(* IEC 61131-3 sources: inproshop/TEAM_V2.0-demo_exported/OP30/2.PRG, 7 files *)

(* ---- OP30_Communication.st ---- *)
PROGRAM OP30_Communication
VAR
	HeartdelayON:TON;
	HeartdelayOFF:TON;
	MasterHeartdelayON:TON;
	MasterHeartdelayOFF:TON;
END_VAR

//心跳输出
IF CPU_Clock.Clock_1s THEN
	DB3005_Communication.TO_OPXX.Heart:=1;
ELSE
	DB3005_Communication.TO_OPXX.Heart:=0;
END_IF
//给前站安全信号
IF TRUE THEN
	DB3005_Communication.TO_OPXX.Safe:=1;
ELSE
	DB3005_Communication.TO_OPXX.Safe:=0;
END_IF;

HeartdelayON(IN:= DB3005_Communication.From_OPXX.Heart=1, PT:= T#2S, Q=> , ET=> );
HeartdelayOFF(IN:= DB3005_Communication.From_OPXX.Heart=0, PT:= T#2S, Q=> , ET=> );
//前站掉线报警
IF (HeartdelayON.Q OR HeartdelayOFF.Q) AND NOT DB3000_Control.Mode.Status.OfflineMode  THEN
	DB3070_Fault.Stop.BeforStation_Communication_Rrror:=TRUE;
END_IF

//主站心跳通讯检测
MasterHeartdelayON(IN:= DB3005_Communication.FromMaster.Heart=1, PT:= T#2S, Q=> , ET=> );
MasterHeartdelayOFF(IN:= DB3005_Communication.FromMaster.Heart=0, PT:= T#2S, Q=> , ET=> );
//主站掉线报警
IF (MasterHeartdelayON.Q OR MasterHeartdelayOFF.Q) AND NOT DB3000_Control.Mode.Status.OfflineMode  THEN
	DB3070_Fault.Stop.MasterTimeOut:=TRUE;
END_IF

//与主站配方不一致报警
IF DB3005_Communication.FromMaster.MasterRecipeID<>DB3002_Recipe.RecipeNum AND NOT DB3000_Control.Mode.Status.OfflineMode THEN
	DB3070_Fault.Stop.MaterReipeDiscrepancy:=TRUE;
END_IF

(* ---- OP30_Control.st ---- *)
PROGRAM OP30_Control
VAR
	FB_ModeControl_instance:FB_ModeControl_V1;
	FB_Count_instance:ARRAY[0..2] OF FB_Count;
END_VAR

(**********模式切换功能***********)
FB_ModeControl_instance(
	iClock:= CPU_Clock,
	iStartDelay:= T#100MS,
	iEstop:=DB3070_Fault.EstopTotal,
	iAlam:=DB3070_Fault.StopTotal,
	iWarn:=DB3070_Fault.RunTotal,
	ioMachine:= DB3000_Control.Machine,
	ioMode:=DB3000_Control.Mode);

(********************计数****************************)
//总计数
FB_Count_instance[0](
	ioCount:= DB3003_Count.Total,
	iClock:= CPU_Clock,
	iDayStartTime:= CPU_Clock.DayStartTime,
	iNightStartTime:=CPU_Clock.NightStartTime);

//OK计数
FB_Count_instance[1](
	ioCount:= DB3003_Count.OK,
	iClock:= CPU_Clock,
	iDayStartTime:= CPU_Clock.DayStartTime,
	iNightStartTime:=CPU_Clock.NightStartTime);

//NG计数
FB_Count_instance[2](
	ioCount:= DB3003_Count.NG,
	iClock:= CPU_Clock,
	iDayStartTime:= CPU_Clock.DayStartTime,
	iNightStartTime:=CPU_Clock.NightStartTime);

(***********良率计算***********)
//良率统计
IF DB3003_Count.Total.Today.Total<>0 THEN
	DB3003_Count.Yield:=DB3003_Count.OK.Today.Total/DB3003_Count.Total.Today.Total;
ELSE
	DB3003_Count.Yield:=0;
END_IF
//良率清零
IF DB3003_Count.Clear THEN
	DB3003_Count.Total.Today.Total:=0;
	DB3003_Count.OK.Today.Total:=0;
	DB3003_Count.NG.Today.Total:=0;
	DB3003_Count.Clear:=FALSE;
END_IF

(********程序调用*******)
OP30_DI_Mirror();
OP30_Communication();
OP30_Recipe();
OP30_Graph();
OP30_DriveControl();
OP30_DO_Mirror();
OP30_Fault();
OP30_Other();

(* ---- OP30_DI_Mirror.st ---- *)
PROGRAM OP30_DI_Mirror
VAR
	i:INT;//循环用变量
	Page:INT;
	Monitor:ARRAY[0..15] OF Str_IOMonitor;
	Status:WORD;
	Map:BOOL;
END_VAR

ACT_MAP();
ACT_Comment();
ACT_Status();

(* ---- OP30_DO_Mirror.st ---- *)
PROGRAM OP30_DO_Mirror
VAR
	i:INT;//循环用变量
	Page:INT;
	Monitor:ARRAY[0..15] OF Str_IOMonitor;
	Status:WORD;
	Map:BOOL;
	Startlamp1:BOOL;
	Startlamp2:BOOL;
END_VAR

ACT_MAP();
ACT_Comment();
ACT_Status();

(* ---- OP30_DriveControl.st ---- *)
PROGRAM OP30_DriveControl
VAR
	FB_Cylinder_instance :ARRAY[0..63]OF FB_Cylinder_V1;
	FB_Vacuum_instance :ARRAY[0..31]OF FB_Vacuum_V1;
	FB_Axis_Instance:ARRAY[0..31]OF FB_Axis_V1_3;
	FB_Sensor_instance :ARRAY[0..200]OF FB_Sensor_V1_1;
	FB_TcpClient_Instance:ARRAY[0..31]OF FB_TcpClient;
	FB_DoubleStart_Instance:ARRAY[1..4]OF FB_DoubleStart;
	FB_Epson_V1_Instance:ARRAY[1..1]OF FB_Epson_V1;
	FB_Kuka_V1_Instance:ARRAY[1..2]OF FB_Kuka6_V1;
	FB_Rotdisk_V1_Instance:ARRAY[1..1]OF FB_Rotdisk_V1;
	FB_Stopper_V1_Instance:ARRAY[1..1]OF FB_Stopper_V1;
	FB_Motor_Instance:ARRAY[1..1]OF FB_Motor;
	FB_Heating_Instance:ARRAY[1..1]OF FB_Heating;
	FB_Gear_Instance:ARRAY[1..1]OF FB_Gear;
	FB_AAS_Instance:ARRAY[1..1]OF FB_AAS;
	FB_AirLeak_Instance:ARRAY[1..2]OF FB_AirLeak;
	FB_Palletizing_Instance:ARRAY[1..3]OF FB_Palletizing;
END_VAR
VAR
	i:INT;//循环变量用
	j:INT;//循环变量用
END_VAR

VAR
	TempKUKA1InPut AT %IB4500:ARRAY[0..63]OF BYTE;
	TempKUKA1OutPut AT %QB4500:ARRAY[0..63]OF BYTE;
	TempKUKA2InPut AT %IB4600:ARRAY[0..63]OF BYTE;
	TempKUKA2OutPut AT %QB4600:ARRAY[0..63]OF BYTE;
END_VAR
VAR
	PowerLimitDelay:ARRAY[0..16] OF TON;//超出额定电流
END_VAR

ACT_Axis();
ACT_Cylinder();
ACT_Vacuum();
ACT_Epson();
ACT_Kuka();
ACT_Sensor();
ACT_Motor();
ACT_Rotdisk();
ACT_AI();
ACT_Stopper();

ACT_Pallet();

(* ---- OP30_Other.st ---- *)
PROGRAM OP30_Other
VAR
	i:INT;//循环变量
	MaterialCode: INT;
END_VAR

(* ---- OP30_Recipe.st ---- *)
PROGRAM OP30_Recipe
VAR
	i:INT;
	DownLoad_R:R_TRIG;
	Download_F:F_TRIG;
	Change:R_TRIG;
END_VAR
VAR RETAIN PERSISTENT
	RecipeNum AT %MB131078 : INT;
END_VAR

//主站一键切换配方
IF To_Slave.OnLineMode=1 THEN
	IF DB3002_Recipe.DownLoad THEN
		To_Slave.RecipeDownLoad:=1;
	ELSE
		To_Slave.RecipeDownLoad:=0;
	END_IF
	To_Slave.RecipeID:=DB3002_Recipe.RecipeNumTemp;
ELSE
	To_Slave.RecipeDownLoad:=0;
END_IF

//配方名
DB3002_Recipe.RecipeName:=DB3002_Recipe.TypeData[DB3002_Recipe.RecipeNum].Name;

//配方参数修改使能
IF DB3002_Recipe.RecipeNum=DB3002_Recipe.RecipeNumTemp THEN
	DB3002_Recipe.ParameterChangePmt:=TRUE;
ELSE
	DB3002_Recipe.ParameterChangePmt:=FALSE;
END_IF

//配方允许切换使能
DB3002_Recipe.RecipeChangePmt:=DB6000_Control.Mode.Status.ManualMode ;

//配方提取
DB3002_Recipe.TypeDataCur:=DB3002_Recipe.TypeData[DB3002_Recipe.RecipeNum];

IF RecipeNum<>DB3002_Recipe.RecipeNumTemp THEN
	DB3002_Recipe.RecipeNameTemp:=DB3002_Recipe.TypeData[DB3002_Recipe.RecipeNumTemp].Name;
	RecipeNum:=DB3002_Recipe.RecipeNumTemp;
END_IF

DownLoad_R(CLK:= DB3002_Recipe.DownLoad);
DownLoad_F(CLK:= DB3002_Recipe.DownLoad);
ACT_Download();
ACT_Upload();
